FUNCTION_BLOCK FB_Alarm
  VAR_INPUT
    Fault_in : BOOL;
    Acknowledge : BOOL;
    Alarm_Reset : BOOL;
  END_VAR
  VAR_OUTPUT
    Active : BOOL;
    Latched : BOOL;
  END_VAR
  VAR
    Acknowledged : BOOL;
  END_VAR

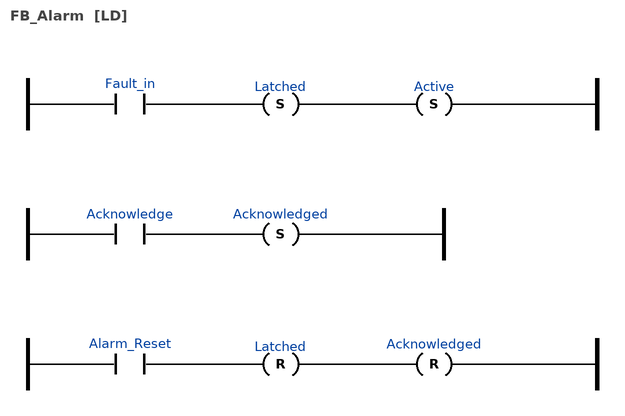
(* LD diagram, written out as Structured Text *)
IF Fault_in THEN Latched := TRUE; END_IF;
IF Fault_in THEN Active := TRUE; END_IF;
IF Acknowledge THEN Acknowledged := TRUE; END_IF;
IF Alarm_Reset THEN Latched := FALSE; END_IF;
IF Alarm_Reset THEN Acknowledged := FALSE; END_IF;
END_FUNCTION_BLOCK
